FUNCTION_BLOCK FB_EcCoESdoWrite
VAR_INPUT
END_VAR
VAR_OUTPUT
END_VAR
VAR
FB_EcCoESdoWriteEx : FB_EcCoESdoWriteEx;

END_VAR

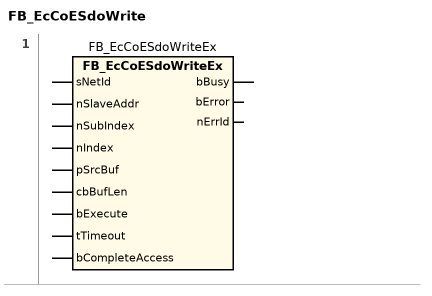
// NETWORK 1
FB_EcCoESdoWriteEx();

END_FUNCTION_BLOCK

(* stored: Version 1.1.0.1, ProductVersion 3.1.4024.12
   POU FB_EcCoESdoWrite: Id {0cfcaf63-6205-47ba-9d76-fc0df2012db7}, SpecialFunc None *)
